Fanuc KAREL source: ka00205.KL

-- PROVISIONAL review KL for V1013-1; original PC SHA256 4154fcba9a259cc2949e7d5cd69e24c6a480e5ff560f5595f9268e70593af00b
-- Incomplete behavior may be omitted. Consult companion uncertainty JSON. Do not deploy.
PROGRAM KA00205
%NOLOCKGROUP
-- UNRESOLVED_DECL SRC type=002013
-- UNRESOLVED_DECL DST type=002013
BEGIN
  -- UNRESOLVED_PC offsets 5-19; opcodes 22,22,1E
  -- UNRESOLVED_PC offsets 24-28; opcodes 7F
END KA00205
